PROGRAM Shutdown1

VAR
	shutdownButton	AT%I* 	:BOOL := TRUE;
	cell1  			AT%I*   :INT:=0;
	cell12 			AT%I*	:INT:=0;
	
	umrechnungSpannung:LREAL:=0.000305185094;
	spannungZelle1:LREAL:=0;
	spannungZelle2:LREAL:=0;
	
	Shutdown_Block: NT_Shutdown;
END_VAR


spannungZelle1:=cell1*umrechnungSpannung;
spannungZelle2 :=(cell1-cell12)*umrechnungSpannung;


IF(spannungZelle1<3.1 OR spannungZelle2 <3.1 OR shutdownButton = FALSE ) THEN
	//Shutdown_Block(DELAY:=3,START:=TRUE);
ELSE
	Shutdown_Block(DELAY:=3,START:=TRUE);
END_IF

END_PROGRAM

(* stored: Version 1.1.0.1, ProductVersion 3.1.4022.3
   POU Shutdown1: Id {0d0a7d0a-6db2-45b6-b6da-063463895a99}, SpecialFunc None *)
